GLOBALCONSTANTS DataPanel_LO_DO (* DataPanel Modules with low IO density DO constants *)
  (* Standard: 61499-1; Description: Copyright (c) 2024 HR Agrartechnik GmbH This program and the accompanying materials are made available under the terms of the Eclipse Public License 2.0 which is available at https://www.eclipse.org/legal/epl-2.0/ SPDX-License-Identifier: EPL-2.0 *)
  (* Version 1.0, 2024-01-25, Franz Höpfinger, HR Agrartechnik GmbH *)
  PACKAGE DataPanel::io::LO::DQ;
  VAR_GLOBAL CONSTANT
    DigitalOutput_1A : DataPanel::io::LO::DQ::DataPanel_LO_DO_S := (Pin := 1);
    DigitalOutput_1B : DataPanel::io::LO::DQ::DataPanel_LO_DO_S := (Pin := 2);
    DigitalOutput_2A : DataPanel::io::LO::DQ::DataPanel_LO_DO_S := (Pin := 3);
    DigitalOutput_2B : DataPanel::io::LO::DQ::DataPanel_LO_DO_S := (Pin := 4);
    DigitalOutput_3A : DataPanel::io::LO::DQ::DataPanel_LO_DO_S := (Pin := 5);
    DigitalOutput_3B : DataPanel::io::LO::DQ::DataPanel_LO_DO_S := (Pin := 6);
    DigitalOutput_4A : DataPanel::io::LO::DQ::DataPanel_LO_DO_S := (Pin := 7);
    DigitalOutput_4B : DataPanel::io::LO::DQ::DataPanel_LO_DO_S := (Pin := 8);
    Invalid : DataPanel::io::LO::DQ::DataPanel_LO_DO_S := (Pin := 255);
  END_VAR
END_GLOBALCONSTANTS
